ADAPTER AdapterCyl (* Adapter Interface *)
  (* Standard: 61499-1 *)
  (* Version 0.0, 7/14/2023, valeriy, nxtControl GmBH *)
  PACKAGE Main;
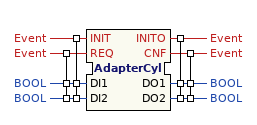
  EVENT_INPUT
    INIT WITH DI1, DI2; (* Request from Socket *)
    REQ WITH DI1, DI2; (* Response from Socket *)
  END_EVENT
  EVENT_OUTPUT
    INITO WITH DO1, DO2; (* Confirmation from Plug *)
    CNF WITH DO1, DO2; (* Indication from Plug *)
  END_EVENT
  VAR_INPUT
    DI1 : BOOL; (* Request Data from Socket *)
    DI2 : BOOL; (* Response Data from Socket *)
  END_VAR
  VAR_OUTPUT
    DO1 : BOOL; (* Confirmation Data from Plug *)
    DO2 : BOOL; (* Indication Data from Plug *)
  END_VAR
  SERVICE SOCKET/PLUG
    SEQUENCE request_confirm
      SOCKET.INIT(DI1) -> PLUG.INIT(DI1);
      PLUG.INITO(DO1) -> SOCKET.INITO(DO1);
    END_SEQUENCE
    SEQUENCE indication_response
      PLUG.CNF(DO2) -> SOCKET.CNF(DO2);
      SOCKET.REQ(DI2) -> PLUG.REQ(DI2);
    END_SEQUENCE
  END_SERVICE
END_ADAPTER
